REGION Network 1: INICIA LEITURA MODBUS
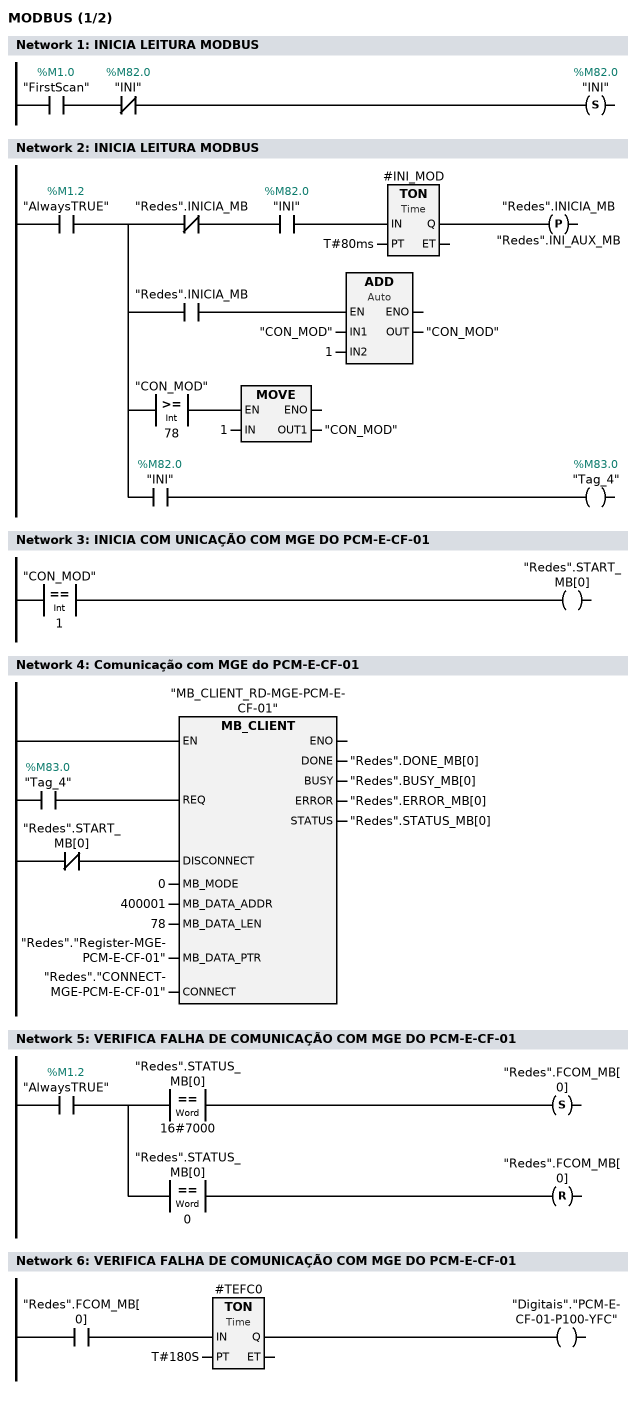
   RUNG wire#powerrail
      Contact( "FirstScan" )
      I_Contact( "INI" )
      S_Coil( "INI" )
   END_RUNG
   // the same network as SCL:
   IF "FirstScan" AND NOT "INI" THEN "INI" := TRUE; END_IF;
END_REGION

REGION Network 2: INICIA LEITURA MODBUS
   #INI_MOD(IN := "AlwaysTRUE" AND NOT "Redes".INICIA_MB AND "INI", PT := T#80ms);   // TON
   "Redes".INICIA_MB := #INI_MOD.Q AND NOT "Redes".INI_AUX_MB;   // rising edge
   "Redes".INI_AUX_MB := #INI_MOD.Q;
   IF "AlwaysTRUE" AND "Redes".INICIA_MB THEN "CON_MOD" := "CON_MOD" + 1; END_IF;
   IF "AlwaysTRUE" AND ("CON_MOD" >= 78) THEN "CON_MOD" := 1; END_IF;
   "Tag_4" := "AlwaysTRUE" AND "INI";
END_REGION

REGION Network 3: INICIA COM UNICAÇÃO COM MGE DO PCM-E-CF-01
   RUNG wire#powerrail
      { S7_Templates := "SrcType := Int" } EQ_Contact(in1 := "CON_MOD", in2 := 1)
      Coil( "Redes".START_MB[0] )
   END_RUNG
   // the same network as SCL:
   "Redes".START_MB[0] := "CON_MOD" = 1;
END_REGION

REGION Network 4: Comunicação com MGE do PCM-E-CF-01
   RUNG wire#powerrail
      "MB_CLIENT_RD-MGE-PCM-E-CF-01".MB_CLIENT(REQ := wire#w1, DISCONNECT := wire#w2, MB_MODE := 0, MB_DATA_ADDR := 400001, MB_DATA_LEN := 78, MB_DATA_PTR := "Redes"."Register-MGE-PCM-E-CF-01", CONNECT := "Redes"."CONNECT-MGE-PCM-E-CF-01", DONE => "Redes".DONE_MB[0], BUSY => "Redes".BUSY_MB[0], ERROR => "Redes".ERROR_MB[0], STATUS => "Redes".STATUS_MB[0])
   END_RUNG
   RUNG wire#powerrail
      Contact( "Tag_4" )
   END_RUNG wire#w1
   RUNG wire#powerrail
      I_Contact( "Redes".START_MB[0] )
   END_RUNG wire#w2
   // the same network as SCL:
   "MB_CLIENT_RD-MGE-PCM-E-CF-01"(REQ := "Tag_4",   // MB_CLIENT
                           DISCONNECT := NOT "Redes".START_MB[0],
                           MB_MODE := 0,
                           MB_DATA_ADDR := 400001,
                           MB_DATA_LEN := 78,
                           MB_DATA_PTR := "Redes"."Register-MGE-PCM-E-CF-01",
                           CONNECT := "Redes"."CONNECT-MGE-PCM-E-CF-01",
                           DONE => "Redes".DONE_MB[0],
                           BUSY => "Redes".BUSY_MB[0],
                           ERROR => "Redes".ERROR_MB[0],
                           STATUS => "Redes".STATUS_MB[0]);
END_REGION

REGION Network 5: VERIFICA FALHA DE COMUNICAÇÃO COM MGE DO PCM-E-CF-01
   RUNG wire#powerrail
      Contact( "AlwaysTRUE" )
      wire#w1
      { S7_Templates := "SrcType := Word" } EQ_Contact(in1 := "Redes".STATUS_MB[0], in2 := 16#7000)
      S_Coil( "Redes".FCOM_MB[0] )
   END_RUNG
   RUNG wire#w1
      { S7_Templates := "SrcType := Word" } EQ_Contact(in1 := "Redes".STATUS_MB[0], in2 := 0)
      R_Coil( "Redes".FCOM_MB[0] )
   END_RUNG
   // the same network as SCL:
   IF "AlwaysTRUE" AND ("Redes".STATUS_MB[0] = 16#7000) THEN "Redes".FCOM_MB[0] := TRUE; END_IF;
   IF "AlwaysTRUE" AND ("Redes".STATUS_MB[0] = 0) THEN "Redes".FCOM_MB[0] := FALSE; END_IF;
END_REGION

REGION Network 6: VERIFICA FALHA DE COMUNICAÇÃO COM MGE DO PCM-E-CF-01
   RUNG wire#powerrail
      Contact( "Redes".FCOM_MB[0] )
      { S7_Templates := "time_type := Time" } #TEFC0.TON(pt := T#180S, et =>)
      Coil( "Digitais"."PCM-E-CF-01-P100-YFC" )
   END_RUNG
   // the same network as SCL:
   #TEFC0(IN := "Redes".FCOM_MB[0], PT := T#180S);   // TON
   "Digitais"."PCM-E-CF-01-P100-YFC" := #TEFC0.Q;
END_REGION

NETWORK
TITLE = Movimentação de dados do MGE PCM-E-CF-01
//CONVERSÃO E MOVIMENTAÇÃO MEDIÇÃO DE TENSÃO
      L     "Redes"."Register-MGE-PCM-E-CF-01"[1];
      DTR;
      L     10.0;
      /R;
      T     "VARIAVEIS"."PCM-E-CF-01-04-P100-ETRS";

      L     "Redes"."Register-MGE-PCM-E-CF-01"[11];
      DTR;
      L     10.0;
      /R;
      T     "VARIAVEIS"."PCM-E-CF-01-04-P100-ETST";

      L     "Redes"."Register-MGE-PCM-E-CF-01"[21];
      DTR;
      L     10.0;
      /R;
      T     "VARIAVEIS"."PCM-E-CF-01-04-P100-ETTR";


//CONVERSÃO E MOVIMENTAÇÃO MEDIÇÃO DE CORRENTE
      L     "Redes"."Register-MGE-PCM-E-CF-01"[2];
      DTR;
      L     100.0;
      /R;
      T     "VARIAVEIS"."PCM-E-CF-01-04-P100-ITR";

      L     "Redes"."Register-MGE-PCM-E-CF-01"[12];
      DTR;
      L     100.0;
      /R;
      T     "VARIAVEIS"."PCM-E-CF-01-04-P100-ITS";

      L     "Redes"."Register-MGE-PCM-E-CF-01"[22];
      DTR;
      L     100.0;
      /R;
      T     "VARIAVEIS"."PCM-E-CF-01-04-P100-ITT";



//CONVERSÃO E MOVIMENTAÇÃO MEDIÇÃO DE POTÊNCIA ATIVA
      L     "Redes"."Register-MGE-PCM-E-CF-01"[34];
      DTR;
      L     100000.0;
      /R;
      T     "VARIAVEIS"."PCM-E-CF-01-04-P100-JPT";

//CONVERSÃO E MOVIMENTAÇÃO MEDIÇÃO DE POTÊNCIA REATIVA
      L     "Redes"."Register-MGE-PCM-E-CF-01"[35];
      DTR;
      L     100000.0;
      /R;
      T     "VARIAVEIS"."PCM-E-CF-01-04-P100-JQT";

//CONVERSÃO E MOVIMENTAÇÃO MEDIÇÃO DE POTÊNCIA APARENTE
      L     "Redes"."Register-MGE-PCM-E-CF-01"[36];
      DTR;
      L     100000.0;
      /R;
      T     "VARIAVEIS"."PCM-E-CF-01-04-P100-JST";

//CONVERSÃO E MOVIMENTAÇÃO MEDIÇÃO DE FATOR DE POTÊNCIA
      L     %DB500.DBW160;
      ITD;
      DTR;
      L     1000.0;
      /R;
      T     "VARIAVEIS"."PCM-E-CF-01-04-P100-FP";



REGION Network 8: INICIA COM UNICAÇÃO COM MGE DO QGBT-AUX-01
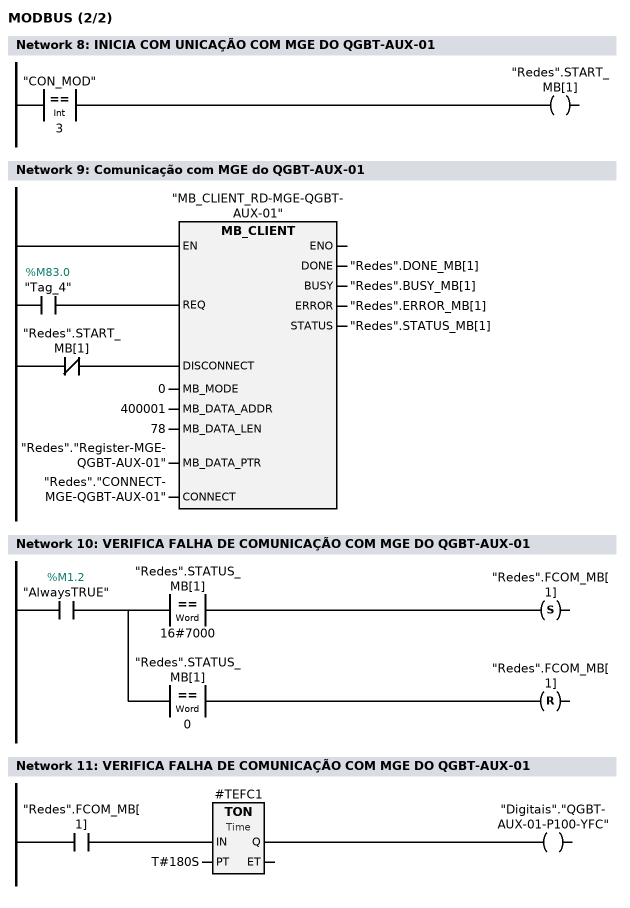
   RUNG wire#powerrail
      { S7_Templates := "SrcType := Int" } EQ_Contact(in1 := "CON_MOD", in2 := 3)
      Coil( "Redes".START_MB[1] )
   END_RUNG
   // the same network as SCL:
   "Redes".START_MB[1] := "CON_MOD" = 3;
END_REGION

REGION Network 9: Comunicação com MGE do QGBT-AUX-01
   RUNG wire#powerrail
      "MB_CLIENT_RD-MGE-QGBT-AUX-01".MB_CLIENT(REQ := wire#w1, DISCONNECT := wire#w2, MB_MODE := 0, MB_DATA_ADDR := 400001, MB_DATA_LEN := 78, MB_DATA_PTR := "Redes"."Register-MGE-QGBT-AUX-01", CONNECT := "Redes"."CONNECT-MGE-QGBT-AUX-01", DONE => "Redes".DONE_MB[1], BUSY => "Redes".BUSY_MB[1], ERROR => "Redes".ERROR_MB[1], STATUS => "Redes".STATUS_MB[1])
   END_RUNG
   RUNG wire#powerrail
      Contact( "Tag_4" )
   END_RUNG wire#w1
   RUNG wire#powerrail
      I_Contact( "Redes".START_MB[1] )
   END_RUNG wire#w2
   // the same network as SCL:
   "MB_CLIENT_RD-MGE-QGBT-AUX-01"(REQ := "Tag_4",   // MB_CLIENT
                           DISCONNECT := NOT "Redes".START_MB[1],
                           MB_MODE := 0,
                           MB_DATA_ADDR := 400001,
                           MB_DATA_LEN := 78,
                           MB_DATA_PTR := "Redes"."Register-MGE-QGBT-AUX-01",
                           CONNECT := "Redes"."CONNECT-MGE-QGBT-AUX-01",
                           DONE => "Redes".DONE_MB[1],
                           BUSY => "Redes".BUSY_MB[1],
                           ERROR => "Redes".ERROR_MB[1],
                           STATUS => "Redes".STATUS_MB[1]);
END_REGION

REGION Network 10: VERIFICA FALHA DE COMUNICAÇÃO COM MGE DO QGBT-AUX-01
   RUNG wire#powerrail
      Contact( "AlwaysTRUE" )
      wire#w1
      { S7_Templates := "SrcType := Word" } EQ_Contact(in1 := "Redes".STATUS_MB[1], in2 := 16#7000)
      S_Coil( "Redes".FCOM_MB[1] )
   END_RUNG
   RUNG wire#w1
      { S7_Templates := "SrcType := Word" } EQ_Contact(in1 := "Redes".STATUS_MB[1], in2 := 0)
      R_Coil( "Redes".FCOM_MB[1] )
   END_RUNG
   // the same network as SCL:
   IF "AlwaysTRUE" AND ("Redes".STATUS_MB[1] = 16#7000) THEN "Redes".FCOM_MB[1] := TRUE; END_IF;
   IF "AlwaysTRUE" AND ("Redes".STATUS_MB[1] = 0) THEN "Redes".FCOM_MB[1] := FALSE; END_IF;
END_REGION

REGION Network 11: VERIFICA FALHA DE COMUNICAÇÃO COM MGE DO QGBT-AUX-01
   RUNG wire#powerrail
      Contact( "Redes".FCOM_MB[1] )
      { S7_Templates := "time_type := Time" } #TEFC1.TON(pt := T#180S, et =>)
      Coil( "Digitais"."QGBT-AUX-01-P100-YFC" )
   END_RUNG
   // the same network as SCL:
   #TEFC1(IN := "Redes".FCOM_MB[1], PT := T#180S);   // TON
   "Digitais"."QGBT-AUX-01-P100-YFC" := #TEFC1.Q;
END_REGION

NETWORK
TITLE = Movimentação de dados do MGE QGBT-AUX-01
//CONVERSÃO E MOVIMENTAÇÃO MEDIÇÃO DE TENSÃO
      L     "Redes"."Register-MGE-QGBT-AUX-01"[1];
      DTR;
      L     10.0;
      /R;
      T     "VARIAVEIS"."QGBT-AUX-01-P100-ETRS";

      L     "Redes"."Register-MGE-QGBT-AUX-01"[11];
      DTR;
      L     10.0;
      /R;
      T     "VARIAVEIS"."QGBT-AUX-01-P100-ETST";

      L     "Redes"."Register-MGE-QGBT-AUX-01"[21];
      DTR;
      L     10.0;
      /R;
      T     "VARIAVEIS"."QGBT-AUX-01-P100-ETTR";


//CONVERSÃO E MOVIMENTAÇÃO MEDIÇÃO DE CORRENTE
      L     "Redes"."Register-MGE-QGBT-AUX-01"[2];
      DTR;
      L     100.0;
      /R;
      T     "VARIAVEIS"."QGBT-AUX-01-P100-ITR";

      L     "Redes"."Register-MGE-QGBT-AUX-01"[12];
      DTR;
      L     100.0;
      /R;
      T     "VARIAVEIS"."QGBT-AUX-01-P100-ITS";

      L     "Redes"."Register-MGE-QGBT-AUX-01"[22];
      DTR;
      L     100.0;
      /R;
      T     "VARIAVEIS"."QGBT-AUX-01-P100-ITT";



//CONVERSÃO E MOVIMENTAÇÃO MEDIÇÃO DE POTÊNCIA ATIVA
      L     "Redes"."Register-MGE-QGBT-AUX-01"[34];
      DTR;
      L     100000.0;
      /R;
      T     "VARIAVEIS"."QGBT-AUX-01-P100-JPT";

//CONVERSÃO E MOVIMENTAÇÃO MEDIÇÃO DE POTÊNCIA REATIVA
      L     "Redes"."Register-MGE-QGBT-AUX-01"[35];
      DTR;
      L     100000.0;
      /R;
      T     "VARIAVEIS"."QGBT-AUX-01-P100-JQT";

//CONVERSÃO E MOVIMENTAÇÃO MEDIÇÃO DE POTÊNCIA APARENTE
      L     "Redes"."Register-MGE-QGBT-AUX-01"[36];
      DTR;
      L     100000.0;
      /R;
      T     "VARIAVEIS"."QGBT-AUX-01-P100-JST";

//CONVERSÃO E MOVIMENTAÇÃO MEDIÇÃO DE FATOR DE POTÊNCIA
      L     %DB500.DBW316;
      ITD;
      DTR;
      L     1000.0;
      /R;
      T     "VARIAVEIS"."QGBT-AUX-01-P100-FP";


END_FUNCTION_BLOCK

FUNCTION_BLOCK "ROD2"   // FB205, LAD
TITLE = RODÍZIO DE 2 GRUPOS
{ S7_Optimized_Access := 'FALSE' }
VERSION : 0.1
// stored: AutoNumber false, IsIECCheckEnabled false, SetENOAutomatically false, UDAEnableTagReadback false
   VAR_INPUT
      G1OK : Bool;   // GRUPO EM CONDIÇÕES DE OPERAÇÃO
      G2OK : Bool;   // GRUPO EM CONDIÇÕES DE OPERAÇÃO
      G1L : Bool;   // GRUPO LIGADO
      G2L : Bool;   // GRUPO LIGADO
      TEROD : Int;   // TEMPOPARA RODÍZIO DAS BOMBAS
      LIGP : Bool;   // LIGA BOMBA PRINCIPAL
      LIGC1 : Bool;   // LIGA BOMBA COMPLEMENTAR 1
      DESAB : Bool;   // DESABILITA FUNCIONAMENTO DOS GRUPOS
      T1S : Bool;   // PULSO A CADA 1 SEGUNDO
      DESAB_PART : Bool;   // DESABILITA RODIZIO POR PARTIDA
   END_VAR
   VAR_OUTPUT
      G1P : Bool;   // GRUPO 1 SELECIONADO COMO PRINCIPAL
      G2P : Bool;   // GRUPO 2 SELECIONADO COMO PRINCIPAL
      G1C1 : Bool;   // GRUPO 1 SELECIONADO COMO COMPLEMENTAR 1
      G2C1 : Bool;   // GRUPO 2 SELECIONADO COMO COMPLEMENTAR 1
      LG1 : Bool;   // LIGA GRUPO 1
      LG2 : Bool;   // LIGA GRUPO 2
   END_VAR
   VAR_IN_OUT
      TOG1P : DInt;   // TEMPO DE OPERAÇÃO GRUPO 1
      TOG2P : DInt;   // TEMPO DE OPERAÇÃO GRUPO 2
      TEOKG1 : Real;   // TEMPO OK GRUPO 1
      TEOKG2 : Real;   // TEMPO OK GRUPO 2
   END_VAR
   VAR DB_SPECIFIC
      GR1SELP : Bool;   // SELECIONADO COMO PRINCIPAL
      GR2SELP : Bool;   // SELECIONADO COMO PRINCIPAL
      GR1SELC1 : Bool;   // SELECIONADO COMO COMPLEMENTAR 1
      GR2SELC1 : Bool;   // SELECIONADO COMO COMPLEMENTAR 1
      PS1SG1 : Bool;   // AUXILIAR DE PULSO
      PS1SG2 : Bool;   // AUXILIAR DE PULSO
      PS1 : Bool;   // AUXILIAR DE PULSO
      PS2 : Bool;   // AUXILIAR DE PULSO
      FIMTEG1 : Bool;   // FIM DO TEMPO DE EXISTÊNCIA DO GRUPO 1
      FIMTEG2 : Bool;   // FIM DO TEMPO DE EXISTÊNCIA DO GRUPO 2
      SDESG1 : Bool;   // SOLICITAÇÃO DE DESLIGAMENTO
      SDESG2 : Bool;   // SOLICITAÇÃO DE DESLIGAMENTO
      GPL : Bool;   // GRUPO PRINCIPAL LIGADO
      GC1L : Bool;   // GRUPO COMPLEMENTAR 1 LIGADO
      SO_L : Bool;   // SOLICITAÇÃO DE PARTIDA
      SO_D : Bool;   // SOLICITAÇÃO DE DESLIGAMENTO
      RTEOPG1 : Bool;   // RESET TEMPO OK
      RTEOPG2 : Bool;   // RESET TEMPO OK
      TON1 { S7_SetPoint := 'True'} : TON_TIME;   // TEMPORIZADOR
      TON2 { S7_SetPoint := 'True'} : TON_TIME;   // TEMPORIZADOR
      TSDG1 { S7_SetPoint := 'True'} : TON_TIME;   // TEMPORIZADOR
      TSDG2 { S7_SetPoint := 'True'} : TON_TIME;   // TEMPORIZADOR
   END_VAR
   VAR_TEMP
      PRI12 : Bool;   // PRIORIDADE GRUPO 1
      TMROD : DInt;   // TEMPO DE RODIZIO
      TEROD_DI : DInt;   // TEMPO DE RODIZIO
      NGS : Int;   // NÚMERO DE GRUPOS SOLICITADOS
      NGF : Int;   // NÚMERO DE GRUPOS FUNCIONANDO
      AUX01 : Int;   // AUXILIAR UTILIZADO NA LÓGICA
      AUX02 : Int;   // AUXILIAR UTILIZADO NA LÓGICA
      AUX03 : Int;   // AUXILIAR UTILIZADO NA LÓGICA
      AUX04 : Int;   // AUXILIAR UTILIZADO NA LÓGICA
      AUX05 : Bool;   // AUXILIAR UTILIZADO NA LÓGICA
      AUX06 : Bool;   // AUXILIAR UTILIZADO NA LÓGICA
      ETT1 : Time;   // EFETIVO DO TEMPORIZADOR
      ETT2 : Time;   // EFETIVO DO TEMPORIZADOR
      ETTSDG2 : Time;   // EFETIVO DO TEMPORIZADOR
      ETTSDG1 : Time;   // EFETIVO DO TEMPORIZADOR
   END_VAR
   VAR_TEMP   // added for the SCL form of the ladder/FBD networks
      _w1 : Bool;
   END_VAR
BEGIN

REGION Network 1: CONVERSÃO DO SETPOINT DE TEMPO DE RODÍZIO
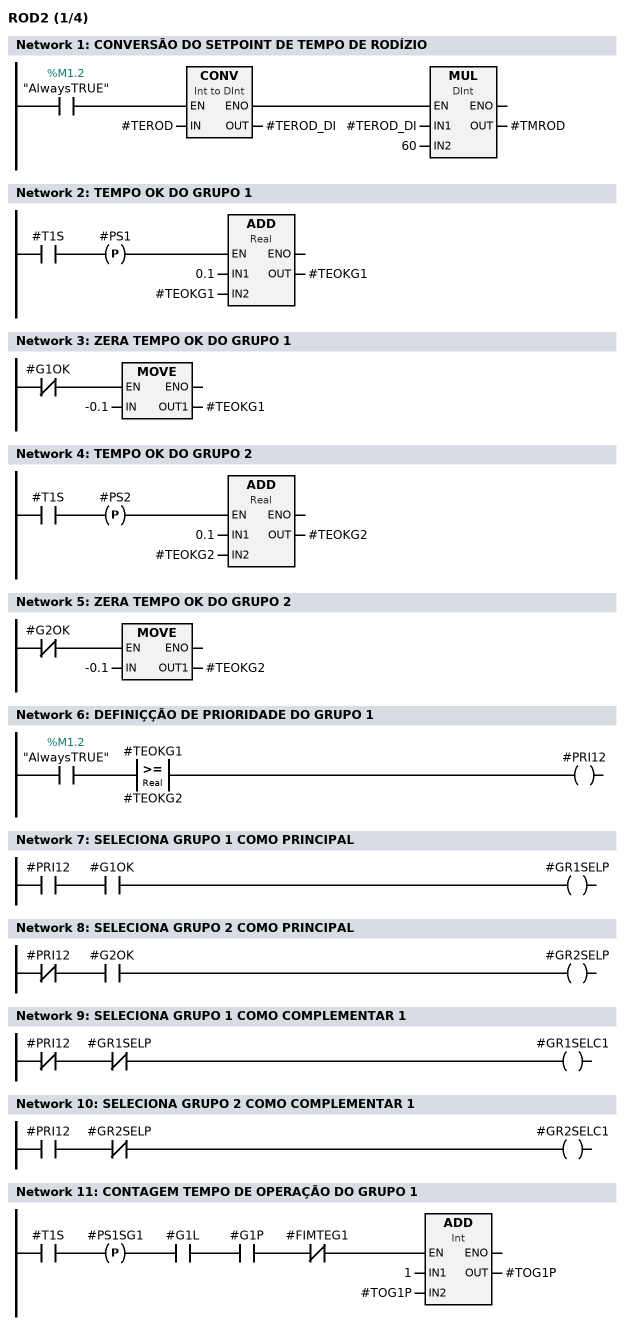
   RUNG wire#powerrail
      Contact( "AlwaysTRUE" )
      { S7_Templates := "[SrcType := Int, DestType := DInt]" } Convert(in := #TEROD, out => #TEROD_DI)
      { S7_Templates := "SrcType := DInt"; S7_GenerateENO := "TRUE" } Mul(in1 := #TEROD_DI, in2 := 60, out => #TMROD)
   END_RUNG
   // the same network as SCL:
   IF "AlwaysTRUE" THEN
       #TEROD_DI := INT_TO_DINT(#TEROD);
       #TMROD := #TEROD_DI * 60;
   END_IF;
END_REGION

REGION Network 2: TEMPO OK DO GRUPO 1
   RUNG wire#powerrail
      Contact( #T1S )
      P_Trig( #PS1 )
      { S7_Templates := "SrcType := Real"; S7_GenerateENO := "TRUE" } Add(in1 := 0.1, in2 := #TEOKG1, out => #TEOKG1)
   END_RUNG
   // the same network as SCL:
   #_w1 := #T1S AND NOT #PS1;   // rising edge
   #PS1 := #T1S;
   IF #_w1 THEN #TEOKG1 := 0.1 + #TEOKG1; END_IF;
END_REGION

REGION Network 3: ZERA TEMPO OK DO GRUPO 1
   RUNG wire#powerrail
      I_Contact( #G1OK )
      { S7_GenerateENO := "TRUE" } Move(in := -0.1, out1 => #TEOKG1)
   END_RUNG
   // the same network as SCL:
   IF NOT #G1OK THEN #TEOKG1 := -0.1; END_IF;
END_REGION

REGION Network 4: TEMPO OK DO GRUPO 2
   RUNG wire#powerrail
      Contact( #T1S )
      P_Trig( #PS2 )
      { S7_Templates := "SrcType := Real"; S7_GenerateENO := "TRUE" } Add(in1 := 0.1, in2 := #TEOKG2, out => #TEOKG2)
   END_RUNG
   // the same network as SCL:
   #_w1 := #T1S AND NOT #PS2;   // rising edge
   #PS2 := #T1S;
   IF #_w1 THEN #TEOKG2 := 0.1 + #TEOKG2; END_IF;
END_REGION

REGION Network 5: ZERA TEMPO OK DO GRUPO 2
   RUNG wire#powerrail
      I_Contact( #G2OK )
      { S7_GenerateENO := "TRUE" } Move(in := -0.1, out1 => #TEOKG2)
   END_RUNG
   // the same network as SCL:
   IF NOT #G2OK THEN #TEOKG2 := -0.1; END_IF;
END_REGION

REGION Network 6: DEFINIÇÇÃO DE PRIORIDADE DO GRUPO 1
   RUNG wire#powerrail
      Contact( "AlwaysTRUE" )
      { S7_Templates := "SrcType := Real" } GE_Contact(in1 := #TEOKG1, in2 := #TEOKG2)
      Coil( #PRI12 )
   END_RUNG
   // the same network as SCL:
   #PRI12 := "AlwaysTRUE" AND (#TEOKG1 >= #TEOKG2);
END_REGION

REGION Network 7: SELECIONA GRUPO 1 COMO PRINCIPAL
   RUNG wire#powerrail
      Contact( #PRI12 )
      Contact( #G1OK )
      Coil( #GR1SELP )
   END_RUNG
   // the same network as SCL:
   #GR1SELP := #PRI12 AND #G1OK;
END_REGION

REGION Network 8: SELECIONA GRUPO 2 COMO PRINCIPAL
   RUNG wire#powerrail
      I_Contact( #PRI12 )
      Contact( #G2OK )
      Coil( #GR2SELP )
   END_RUNG
   // the same network as SCL:
   #GR2SELP := NOT #PRI12 AND #G2OK;
END_REGION

REGION Network 9: SELECIONA GRUPO 1 COMO COMPLEMENTAR 1
   RUNG wire#powerrail
      I_Contact( #PRI12 )
      I_Contact( #GR1SELP )
      Coil( #GR1SELC1 )
   END_RUNG
   // the same network as SCL:
   #GR1SELC1 := NOT #PRI12 AND NOT #GR1SELP;
END_REGION

REGION Network 10: SELECIONA GRUPO 2 COMO COMPLEMENTAR 1
   RUNG wire#powerrail
      Contact( #PRI12 )
      I_Contact( #GR2SELP )
      Coil( #GR2SELC1 )
   END_RUNG
   // the same network as SCL:
   #GR2SELC1 := #PRI12 AND NOT #GR2SELP;
END_REGION

REGION Network 11: CONTAGEM TEMPO DE OPERAÇÃO DO GRUPO 1
   RUNG wire#powerrail
      Contact( #T1S )
      P_Trig( #PS1SG1 )
      Contact( #G1L )
      Contact( #G1P )
      I_Contact( #FIMTEG1 )
      { S7_Templates := "SrcType := Int"; S7_GenerateENO := "TRUE" } Add(in1 := 1, in2 := #TOG1P, out => #TOG1P)
   END_RUNG
   // the same network as SCL:
   #_w1 := #T1S AND NOT #PS1SG1;   // rising edge
   #PS1SG1 := #T1S;
   IF #_w1 AND #G1L AND #G1P AND NOT #FIMTEG1 THEN #TOG1P := 1 + #TOG1P; END_IF;
END_REGION

REGION Network 12: TEMPO DE OPERAÇÃO ATINGIDO
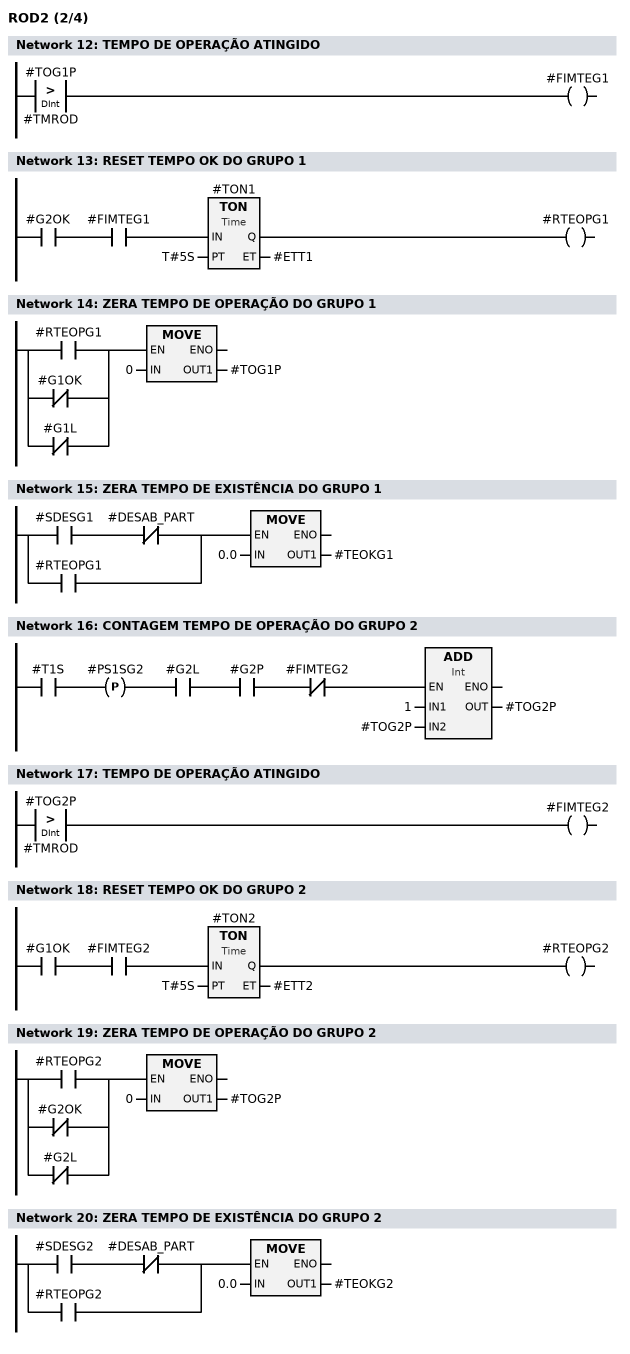
   RUNG wire#powerrail
      { S7_Templates := "SrcType := DInt" } GT_Contact(in1 := #TOG1P, in2 := #TMROD)
      Coil( #FIMTEG1 )
   END_RUNG
   // the same network as SCL:
   #FIMTEG1 := #TOG1P > #TMROD;
END_REGION

REGION Network 13: RESET TEMPO OK DO GRUPO 1
   RUNG wire#powerrail
      Contact( #G2OK )
      Contact( #FIMTEG1 )
      { S7_Templates := "time_type := Time" } #TON1.TON(pt := T#5S, et => #ETT1)
      Coil( #RTEOPG1 )
   END_RUNG
   // the same network as SCL:
   #TON1(IN := #G2OK AND #FIMTEG1, PT := T#5S, ET => #ETT1);   // TON
   #RTEOPG1 := #TON1.Q;
END_REGION

REGION Network 14: ZERA TEMPO DE OPERAÇÃO DO GRUPO 1
   RUNG wire#powerrail
      Contact( #RTEOPG1 )
      wire#w1
      { S7_GenerateENO := "TRUE" } Move(in := 0, out1 => #TOG1P)
   END_RUNG
   RUNG wire#powerrail
      I_Contact( #G1OK )
   END_RUNG wire#w1
   RUNG wire#powerrail
      I_Contact( #G1L )
   END_RUNG wire#w1
   // the same network as SCL:
   IF #RTEOPG1 OR NOT #G1OK OR NOT #G1L THEN #TOG1P := 0; END_IF;
END_REGION

REGION Network 15: ZERA TEMPO DE EXISTÊNCIA DO GRUPO 1
   RUNG wire#powerrail
      Contact( #SDESG1 )
      I_Contact( #DESAB_PART )
      wire#w1
      { S7_GenerateENO := "TRUE" } Move(in := 0.0, out1 => #TEOKG1)
   END_RUNG
   RUNG wire#powerrail
      Contact( #RTEOPG1 )
   END_RUNG wire#w1
   // the same network as SCL:
   IF (#SDESG1 AND NOT #DESAB_PART) OR #RTEOPG1 THEN #TEOKG1 := 0.0; END_IF;
END_REGION

REGION Network 16: CONTAGEM TEMPO DE OPERAÇÃO DO GRUPO 2
   RUNG wire#powerrail
      Contact( #T1S )
      P_Trig( #PS1SG2 )
      Contact( #G2L )
      Contact( #G2P )
      I_Contact( #FIMTEG2 )
      { S7_Templates := "SrcType := Int"; S7_GenerateENO := "TRUE" } Add(in1 := 1, in2 := #TOG2P, out => #TOG2P)
   END_RUNG
   // the same network as SCL:
   #_w1 := #T1S AND NOT #PS1SG2;   // rising edge
   #PS1SG2 := #T1S;
   IF #_w1 AND #G2L AND #G2P AND NOT #FIMTEG2 THEN #TOG2P := 1 + #TOG2P; END_IF;
END_REGION

REGION Network 17: TEMPO DE OPERAÇÃO ATINGIDO
   RUNG wire#powerrail
      { S7_Templates := "SrcType := DInt" } GT_Contact(in1 := #TOG2P, in2 := #TMROD)
      Coil( #FIMTEG2 )
   END_RUNG
   // the same network as SCL:
   #FIMTEG2 := #TOG2P > #TMROD;
END_REGION

REGION Network 18: RESET TEMPO OK DO GRUPO 2
   RUNG wire#powerrail
      Contact( #G1OK )
      Contact( #FIMTEG2 )
      { S7_Templates := "time_type := Time" } #TON2.TON(pt := T#5S, et => #ETT2)
      Coil( #RTEOPG2 )
   END_RUNG
   // the same network as SCL:
   #TON2(IN := #G1OK AND #FIMTEG2, PT := T#5S, ET => #ETT2);   // TON
   #RTEOPG2 := #TON2.Q;
END_REGION

REGION Network 19: ZERA TEMPO DE OPERAÇÃO DO GRUPO 2
   RUNG wire#powerrail
      Contact( #RTEOPG2 )
      wire#w1
      { S7_GenerateENO := "TRUE" } Move(in := 0, out1 => #TOG2P)
   END_RUNG
   RUNG wire#powerrail
      I_Contact( #G2OK )
   END_RUNG wire#w1
   RUNG wire#powerrail
      I_Contact( #G2L )
   END_RUNG wire#w1
   // the same network as SCL:
   IF #RTEOPG2 OR NOT #G2OK OR NOT #G2L THEN #TOG2P := 0; END_IF;
END_REGION

REGION Network 20: ZERA TEMPO DE EXISTÊNCIA DO GRUPO 2
   RUNG wire#powerrail
      Contact( #SDESG2 )
      I_Contact( #DESAB_PART )
      wire#w1
      { S7_GenerateENO := "TRUE" } Move(in := 0.0, out1 => #TEOKG2)
   END_RUNG
   RUNG wire#powerrail
      Contact( #RTEOPG2 )
   END_RUNG wire#w1
   // the same network as SCL:
   IF (#SDESG2 AND NOT #DESAB_PART) OR #RTEOPG2 THEN #TEOKG2 := 0.0; END_IF;
END_REGION

REGION Network 21: SELEÇÃO GRUPO 1 COMO PRINCIPAL
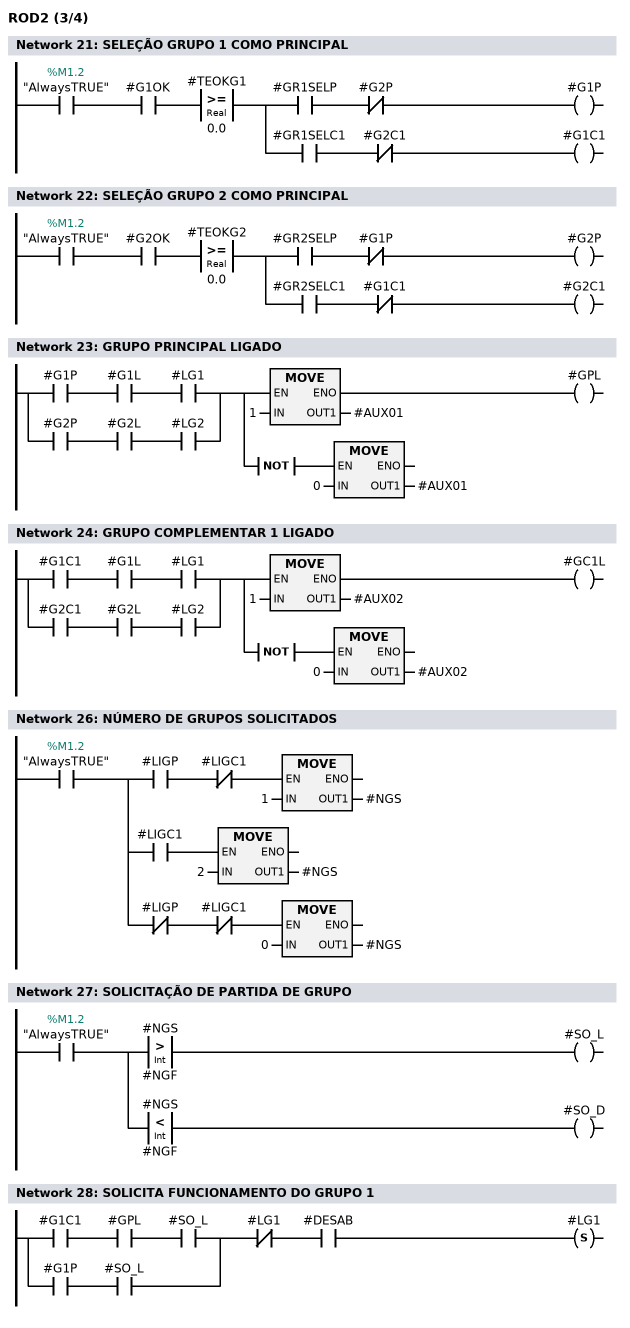
   RUNG wire#powerrail
      Contact( "AlwaysTRUE" )
      Contact( #G1OK )
      { S7_Templates := "SrcType := Real" } GE_Contact(in1 := #TEOKG1, in2 := 0.0)
      wire#w1
      Contact( #GR1SELP )
      I_Contact( #G2P )
      Coil( #G1P )
   END_RUNG
   RUNG wire#w1
      Contact( #GR1SELC1 )
      I_Contact( #G2C1 )
      Coil( #G1C1 )
   END_RUNG
   // the same network as SCL:
   #_w1 := "AlwaysTRUE" AND #G1OK AND (#TEOKG1 >= 0.0);
   #G1P := #_w1 AND #GR1SELP AND NOT #G2P;
   #G1C1 := #_w1 AND #GR1SELC1 AND NOT #G2C1;
END_REGION

REGION Network 22: SELEÇÃO GRUPO 2 COMO PRINCIPAL
   RUNG wire#powerrail
      Contact( "AlwaysTRUE" )
      Contact( #G2OK )
      { S7_Templates := "SrcType := Real" } GE_Contact(in1 := #TEOKG2, in2 := 0.0)
      wire#w1
      Contact( #GR2SELP )
      I_Contact( #G1P )
      Coil( #G2P )
   END_RUNG
   RUNG wire#w1
      Contact( #GR2SELC1 )
      I_Contact( #G1C1 )
      Coil( #G2C1 )
   END_RUNG
   // the same network as SCL:
   #_w1 := "AlwaysTRUE" AND #G2OK AND (#TEOKG2 >= 0.0);
   #G2P := #_w1 AND #GR2SELP AND NOT #G1P;
   #G2C1 := #_w1 AND #GR2SELC1 AND NOT #G1C1;
END_REGION

REGION Network 23: GRUPO PRINCIPAL LIGADO
   RUNG wire#powerrail
      Contact( #G1P )
      Contact( #G1L )
      Contact( #LG1 )
      wire#w1
      { S7_GenerateENO := "TRUE" } Move(in := 1, out1 => #AUX01)
      Coil( #GPL )
   END_RUNG
   RUNG wire#powerrail
      Contact( #G2P )
      Contact( #G2L )
      Contact( #LG2 )
   END_RUNG wire#w1
   RUNG wire#w1
      Not()
      { S7_GenerateENO := "TRUE" } Move(in := 0, out1 => #AUX01)
   END_RUNG
   // the same network as SCL:
   // ENO of a box is taken as its EN; it also drops when the box reports an error
   #_w1 := (#G1P AND #G1L AND #LG1) OR (#G2P AND #G2L AND #LG2);
   IF #_w1 THEN #AUX01 := 1; END_IF;
   #GPL := #_w1;
   IF NOT #_w1 THEN #AUX01 := 0; END_IF;
END_REGION

REGION Network 24: GRUPO COMPLEMENTAR 1 LIGADO
   RUNG wire#powerrail
      Contact( #G1C1 )
      Contact( #G1L )
      Contact( #LG1 )
      wire#w1
      { S7_GenerateENO := "TRUE" } Move(in := 1, out1 => #AUX02)
      Coil( #GC1L )
   END_RUNG
   RUNG wire#powerrail
      Contact( #G2C1 )
      Contact( #G2L )
      Contact( #LG2 )
   END_RUNG wire#w1
   RUNG wire#w1
      Not()
      { S7_GenerateENO := "TRUE" } Move(in := 0, out1 => #AUX02)
   END_RUNG
   // the same network as SCL:
   // ENO of a box is taken as its EN; it also drops when the box reports an error
   #_w1 := (#G1C1 AND #G1L AND #LG1) OR (#G2C1 AND #G2L AND #LG2);
   IF #_w1 THEN #AUX02 := 1; END_IF;
   #GC1L := #_w1;
   IF NOT #_w1 THEN #AUX02 := 0; END_IF;
END_REGION

NETWORK
TITLE = NÚMERO DE GRUPOS FUNCIONANDO

      L     #AUX01;
      L     #AUX02;
      +I;
      T     #NGF;

REGION Network 26: NÚMERO DE GRUPOS SOLICITADOS
   RUNG wire#powerrail
      Contact( "AlwaysTRUE" )
      wire#w1
      Contact( #LIGP )
      I_Contact( #LIGC1 )
      { S7_GenerateENO := "TRUE" } Move(in := 1, out1 => #NGS)
   END_RUNG
   RUNG wire#w1
      Contact( #LIGC1 )
      { S7_GenerateENO := "TRUE" } Move(in := 2, out1 => #NGS)
   END_RUNG
   RUNG wire#w1
      I_Contact( #LIGP )
      I_Contact( #LIGC1 )
      { S7_GenerateENO := "TRUE" } Move(in := 0, out1 => #NGS)
   END_RUNG
   // the same network as SCL:
   IF "AlwaysTRUE" AND #LIGP AND NOT #LIGC1 THEN #NGS := 1; END_IF;
   IF "AlwaysTRUE" AND #LIGC1 THEN #NGS := 2; END_IF;
   IF "AlwaysTRUE" AND NOT #LIGP AND NOT #LIGC1 THEN #NGS := 0; END_IF;
END_REGION

REGION Network 27: SOLICITAÇÃO DE PARTIDA DE GRUPO
   RUNG wire#powerrail
      Contact( "AlwaysTRUE" )
      wire#w1
      { S7_Templates := "SrcType := Int" } GT_Contact(in1 := #NGS, in2 := #NGF)
      Coil( #SO_L )
   END_RUNG
   RUNG wire#w1
      { S7_Templates := "SrcType := Int" } LT_Contact(in1 := #NGS, in2 := #NGF)
      Coil( #SO_D )
   END_RUNG
   // the same network as SCL:
   #SO_L := "AlwaysTRUE" AND (#NGS > #NGF);
   #SO_D := "AlwaysTRUE" AND (#NGS < #NGF);
END_REGION

REGION Network 28: SOLICITA FUNCIONAMENTO DO GRUPO 1
   RUNG wire#powerrail
      Contact( #G1C1 )
      Contact( #GPL )
      Contact( #SO_L )
      wire#w1
      I_Contact( #LG1 )
      Contact( #DESAB )
      S_Coil( #LG1 )
   END_RUNG
   RUNG wire#powerrail
      Contact( #G1P )
      Contact( #SO_L )
   END_RUNG wire#w1
   // the same network as SCL:
   IF ((#G1C1 AND #GPL AND #SO_L) OR (#G1P AND #SO_L)) AND NOT #LG1 AND #DESAB THEN #LG1 := TRUE; END_IF;
END_REGION

REGION Network 29: SOLICITA FUNCIONAMENTO DO GRUPO 2
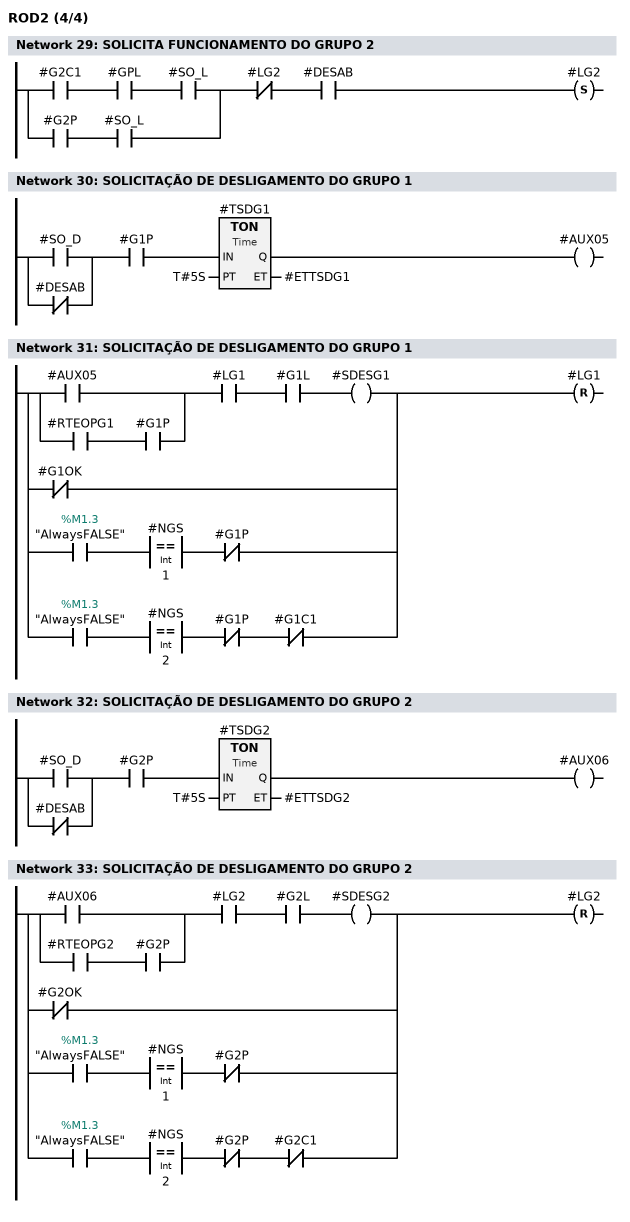
   RUNG wire#powerrail
      Contact( #G2C1 )
      Contact( #GPL )
      Contact( #SO_L )
      wire#w1
      I_Contact( #LG2 )
      Contact( #DESAB )
      S_Coil( #LG2 )
   END_RUNG
   RUNG wire#powerrail
      Contact( #G2P )
      Contact( #SO_L )
   END_RUNG wire#w1
   // the same network as SCL:
   IF ((#G2C1 AND #GPL AND #SO_L) OR (#G2P AND #SO_L)) AND NOT #LG2 AND #DESAB THEN #LG2 := TRUE; END_IF;
END_REGION

REGION Network 30: SOLICITAÇÃO DE DESLIGAMENTO DO GRUPO 1
   RUNG wire#powerrail
      Contact( #SO_D )
      wire#w1
      Contact( #G1P )
      { S7_Templates := "time_type := Time" } #TSDG1.TON(pt := T#5S, et => #ETTSDG1)
      Coil( #AUX05 )
   END_RUNG
   RUNG wire#powerrail
      I_Contact( #DESAB )
   END_RUNG wire#w1
   // the same network as SCL:
   #TSDG1(IN := (#SO_D OR NOT #DESAB) AND #G1P, PT := T#5S, ET => #ETTSDG1);   // TON
   #AUX05 := #TSDG1.Q;
END_REGION

REGION Network 31: SOLICITAÇÃO DE DESLIGAMENTO DO GRUPO 1
   RUNG wire#powerrail
      Contact( #AUX05 )
      wire#w1
      Contact( #LG1 )
      Contact( #G1L )
      Coil( #SDESG1 )
      wire#w2
      R_Coil( #LG1 )
   END_RUNG
   RUNG wire#powerrail
      Contact( #RTEOPG1 )
      Contact( #G1P )
   END_RUNG wire#w1
   RUNG wire#powerrail
      I_Contact( #G1OK )
   END_RUNG wire#w2
   RUNG wire#powerrail
      Contact( "AlwaysFALSE" )
      { S7_Templates := "SrcType := Int" } EQ_Contact(in1 := #NGS, in2 := 1)
      I_Contact( #G1P )
   END_RUNG wire#w2
   RUNG wire#powerrail
      Contact( "AlwaysFALSE" )
      { S7_Templates := "SrcType := Int" } EQ_Contact(in1 := #NGS, in2 := 2)
      I_Contact( #G1P )
      I_Contact( #G1C1 )
   END_RUNG wire#w2
   // the same network as SCL:
   #SDESG1 := (#AUX05 OR (#RTEOPG1 AND #G1P)) AND #LG1 AND #G1L;
   IF #SDESG1 OR NOT #G1OK OR ("AlwaysFALSE" AND (#NGS = 1) AND NOT #G1P) OR ("AlwaysFALSE" AND (#NGS = 2) AND NOT #G1P AND NOT #G1C1) THEN
       #LG1 := FALSE;
   END_IF;
END_REGION

REGION Network 32: SOLICITAÇÃO DE DESLIGAMENTO DO GRUPO 2
   RUNG wire#powerrail
      Contact( #SO_D )
      wire#w1
      Contact( #G2P )
      { S7_Templates := "time_type := Time" } #TSDG2.TON(pt := T#5S, et => #ETTSDG2)
      Coil( #AUX06 )
   END_RUNG
   RUNG wire#powerrail
      I_Contact( #DESAB )
   END_RUNG wire#w1
   // the same network as SCL:
   #TSDG2(IN := (#SO_D OR NOT #DESAB) AND #G2P, PT := T#5S, ET => #ETTSDG2);   // TON
   #AUX06 := #TSDG2.Q;
END_REGION

REGION Network 33: SOLICITAÇÃO DE DESLIGAMENTO DO GRUPO 2
   RUNG wire#powerrail
      Contact( #AUX06 )
      wire#w1
      Contact( #LG2 )
      Contact( #G2L )
      Coil( #SDESG2 )
      wire#w2
      R_Coil( #LG2 )
   END_RUNG
   RUNG wire#powerrail
      Contact( #RTEOPG2 )
      Contact( #G2P )
   END_RUNG wire#w1
   RUNG wire#powerrail
      I_Contact( #G2OK )
   END_RUNG wire#w2
   RUNG wire#powerrail
      Contact( "AlwaysFALSE" )
      { S7_Templates := "SrcType := Int" } EQ_Contact(in1 := #NGS, in2 := 1)
      I_Contact( #G2P )
   END_RUNG wire#w2
   RUNG wire#powerrail
      Contact( "AlwaysFALSE" )
      { S7_Templates := "SrcType := Int" } EQ_Contact(in1 := #NGS, in2 := 2)
      I_Contact( #G2P )
      I_Contact( #G2C1 )
   END_RUNG wire#w2
   // the same network as SCL:
   #SDESG2 := (#AUX06 OR (#RTEOPG2 AND #G2P)) AND #LG2 AND #G2L;
   IF #SDESG2 OR NOT #G2OK OR ("AlwaysFALSE" AND (#NGS = 1) AND NOT #G2P) OR ("AlwaysFALSE" AND (#NGS = 2) AND NOT #G2P AND NOT #G2C1) THEN
       #LG2 := FALSE;
   END_IF;
END_REGION
END_FUNCTION_BLOCK

DATA_BLOCK "ANALOGICOS_DB"   // DB101
VERSION : 0.1
// stored: AutoNumber false, DBAccessibleFromOPCUA true, InstanceOfName ANALOGICOS, InstanceOfType FB
"ANALOGICOS"
BEGIN
END_DATA_BLOCK

DATA_BLOCK "INTPRO_DB"   // DB2
VERSION : 0.1
// stored: AutoNumber true, DBAccessibleFromOPCUA true, InstanceOfName INTPRO, InstanceOfType FB
"INTPRO"
BEGIN
END_DATA_BLOCK

DATA_BLOCK "LOOP_DB"   // DB3
VERSION : 0.1
// stored: AutoNumber true, DBAccessibleFromOPCUA true, InstanceOfName LOOP, InstanceOfType FB
"LOOP"
BEGIN
END_DATA_BLOCK

DATA_BLOCK "MODBUS_DB"   // DB102
VERSION : 0.1
// stored: AutoNumber false, DBAccessibleFromOPCUA true, InstanceOfName MODBUS, InstanceOfType FB
"MODBUS"
BEGIN
END_DATA_BLOCK

DATA_BLOCK "PDIR_DB_MB-01"   // DB422
VERSION : 0.1
// stored: AutoNumber false, DBAccessibleFromOPCUA true, InstanceOfName PDIR, InstanceOfType FB
"PDIR"
BEGIN
END_DATA_BLOCK

DATA_BLOCK "PDIR_DB_MB-02"   // DB423
VERSION : 0.1
// stored: AutoNumber false, DBAccessibleFromOPCUA true, InstanceOfName PDIR, InstanceOfType FB
"PDIR"
BEGIN
END_DATA_BLOCK

DATA_BLOCK "PDIR_DB_MB-03"   // DB424
VERSION : 0.1
// stored: AutoNumber false, DBAccessibleFromOPCUA true, InstanceOfName PDIR, InstanceOfType FB
"PDIR"
BEGIN
END_DATA_BLOCK

DATA_BLOCK "PDIR_DB_MB-04"   // DB425
VERSION : 0.1
// stored: AutoNumber false, DBAccessibleFromOPCUA true, InstanceOfName PDIR, InstanceOfType FB
"PDIR"
BEGIN
END_DATA_BLOCK

DATA_BLOCK "ROD4_DB"   // DB9
VERSION : 0.1
// stored: AutoNumber true, DBAccessibleFromOPCUA true, InstanceOfName ROD4, InstanceOfType FB
"ROD4"
BEGIN
END_DATA_BLOCK

DATA_BLOCK "MB_CLIENT_RD-MGE-PCM-E-CF-01"   // DB501
// stored: AutoNumber true, DBAccessibleFromOPCUA true, InstanceOfName MB_CLIENT_1, OfSystemLibElement MB_CLIENT, OfSystemLibVersion 5.1
"MB_CLIENT_1"
   // VAR_INPUT
   //    REQ : Bool;
   //    DISCONNECT : Bool;
   //    MB_MODE : USInt;
   //    MB_DATA_ADDR : UDInt;
   //    MB_DATA_LEN : UInt;
   // END_VAR
   // VAR_OUTPUT
   //    DONE : Bool;
   //    BUSY : Bool;
   //    ERROR : Bool;
   //    STATUS { ExternalVisible := 'False'} : Word;
   // END_VAR
   // VAR_IN_OUT
   //    MB_DATA_PTR : Variant;
   //    CONNECT : Variant;
   // END_VAR
   // VAR
   //    TCON { S7_SetPoint := 'True'} : TCON;
   //    TDISCON { S7_SetPoint := 'True'} : TDISCON;
   //    TSEND { S7_SetPoint := 'True'} : TSEND;
   //    TRECEIVE { S7_SetPoint := 'True'} : TRCV;
   //    TRESET { S7_SetPoint := 'True'} : T_RESET;
   //    TDIAG { S7_SetPoint := 'True'} : T_DIAG;
   //    TDIAG_Status { S7_SetPoint := 'True'} : TDiag_Status;
   //    Blocked_Proc_Timeout : Real;
   //    Rcv_Timeout : Real;
   //    MB_Unit_ID : Byte;
   //    MB_Transaction_ID : Word;
   //    MB_State { ExternalWritable := 'False'} : Word;
   //    SAVED_MB_DATA_ADDR : UDInt;
   //    SAVED_DATA_LEN : UInt;
   //    SAVED_MB_MODE : USInt;
   //    Connection_ID : Word;
   //    Retries : Word;
   //    TEMP_DATA { ExternalWritable := 'False'} : Array[1..263] of Byte;
   //    rcv_timer { ExternalAccessible := 'False'; ExternalVisible := 'False'; ExternalWritable := 'False'; S7_SetPoint := 'True'} : TON_TIME;
   //    wd_timer { ExternalAccessible := 'False'; ExternalVisible := 'False'; ExternalWritable := 'False'; S7_SetPoint := 'True'} : TON_TIME;
   //    Connected : Bool;
   //    Active { ExternalWritable := 'False'} : Bool;
   // END_VAR
BEGIN
END_DATA_BLOCK

DATA_BLOCK "MB_CLIENT_RD-MGE-QGBT-AUX-01"   // DB4
// stored: AutoNumber true, DBAccessibleFromOPCUA true, InstanceOfName MB_CLIENT_1, OfSystemLibElement MB_CLIENT, OfSystemLibVersion 5.1
"MB_CLIENT_1"
   // VAR_INPUT
   //    REQ : Bool;
   //    DISCONNECT : Bool;
   //    MB_MODE : USInt;
   //    MB_DATA_ADDR : UDInt;
   //    MB_DATA_LEN : UInt;
   // END_VAR
   // VAR_OUTPUT
   //    DONE : Bool;
   //    BUSY : Bool;
   //    ERROR : Bool;
   //    STATUS { ExternalVisible := 'False'} : Word;
   // END_VAR
   // VAR_IN_OUT
   //    MB_DATA_PTR : Variant;
   //    CONNECT : Variant;
   // END_VAR
   // VAR
   //    TCON { S7_SetPoint := 'True'} : TCON;
   //    TDISCON { S7_SetPoint := 'True'} : TDISCON;
   //    TSEND { S7_SetPoint := 'True'} : TSEND;
   //    TRECEIVE { S7_SetPoint := 'True'} : TRCV;
   //    TRESET { S7_SetPoint := 'True'} : T_RESET;
   //    TDIAG { S7_SetPoint := 'True'} : T_DIAG;
   //    TDIAG_Status { S7_SetPoint := 'True'} : TDiag_Status;
   //    Blocked_Proc_Timeout : Real;
   //    Rcv_Timeout : Real;
   //    MB_Unit_ID : Byte;
   //    MB_Transaction_ID : Word;
   //    MB_State { ExternalWritable := 'False'} : Word;
   //    SAVED_MB_DATA_ADDR : UDInt;
   //    SAVED_DATA_LEN : UInt;
   //    SAVED_MB_MODE : USInt;
   //    Connection_ID : Word;
   //    Retries : Word;
   //    TEMP_DATA { ExternalWritable := 'False'} : Array[1..263] of Byte;
   //    rcv_timer { ExternalAccessible := 'False'; ExternalVisible := 'False'; ExternalWritable := 'False'; S7_SetPoint := 'True'} : TON_TIME;
   //    wd_timer { ExternalAccessible := 'False'; ExternalVisible := 'False'; ExternalWritable := 'False'; S7_SetPoint := 'True'} : TON_TIME;
   //    Connected : Bool;
   //    Active { ExternalWritable := 'False'} : Bool;
   // END_VAR
BEGIN
END_DATA_BLOCK
